(* CoDeSys 2.3.9.52 project: TrafficLights_pedeX_v1.pro *)
(* Libraries: STANDARD.LIB 16.8.17 14:08:57 *)

(* Global variable list: Global_Variables *)
VAR_GLOBAL
	I_S1		: BOOL; (*Pedestrian X button North*)
	I_S2		: BOOL; (*Pedestrian X button South*)
	O_L1_N_Red	: BOOL; (*Light red, Pedestrian North-South*)
	O_L3_N_Grn	: BOOL;	(*Light green, Pedestrian North-South*)
	O_L4_E_Red	: BOOL;	(*Light red, Cars East-West*)
	O_L5_E_Yel	: BOOL;	(*Light yellow, Cars East-West*)
	O_L6_E_Grn  	: BOOL;	(*Light green, Cars East-West*)
END_VAR

(* POU PRG_BlinkingSimple, ST *)
PROGRAM PRG_BlinkingSimple
(*Niko Siltala
Avustavia laskentaoperaatioita
- vilkutussignaalit
*)
VAR_OUTPUT
	bSign1Hz:BOOL;					(*1 Hz (60krt/min) taajudella vaihteleva signaali*)
END_VAR
VAR
	bInitDone	: BOOL	:=FALSE;	(*Ohjelman initialisointi*)
	c : INT	:=0;				(*Blink counter*)
END_VAR
(*Ohjelman initialisoinnit - Suoritetaan vain kertaalleen*)
IF NOT bInitDone THEN
	bInitDone := TRUE;
END_IF;

(*Making 1Hz blinking signal in case of simulator*)
CASE c OF
0:
	bSign1Hz:= TRUE;
1:
	bSign1Hz:= FALSE;
ELSE
	bSign1Hz:= FALSE;
END_CASE;

(*Add counter *)
c:= c + 1;
IF c > 1 THEN
	c := 0;
END_IF;
END_PROGRAM

(* POU SFC_StateModel, SFC *)
PROGRAM SFC_StateModel
VAR
	tDelay	: TIME	:= T#1s;
	tDelay_Walk : TIME := T#5s;
	srPedestrianReq	: SR;	(*Request from pedestrians has arrived*)
END_VAR
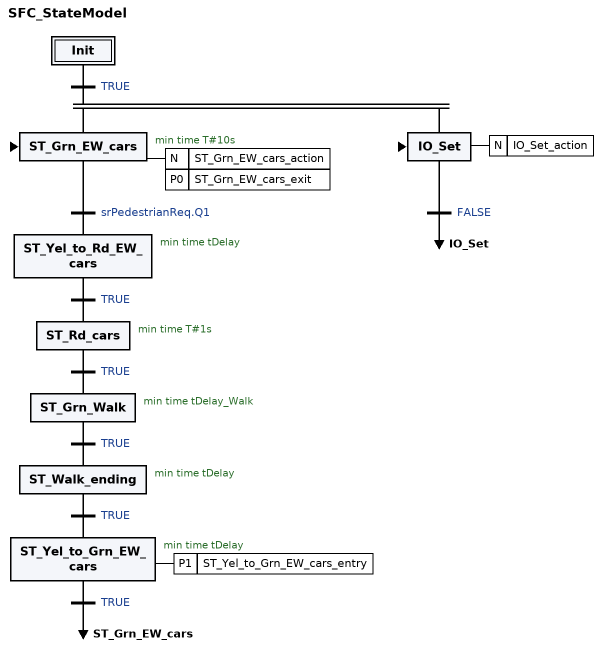
INITIAL_STEP Init:
END_STEP
TRANSITION FROM Init TO (ST_Grn_EW_cars, IO_Set) := TRUE;
END_TRANSITION
STEP ST_Grn_EW_cars: (* min time T#10s *)
	ST_Grn_EW_cars_action(N);
	ST_Grn_EW_cars_exit(P0);
END_STEP
TRANSITION FROM ST_Grn_EW_cars TO ST_Yel_to_Rd_EW_cars := srPedestrianReq.Q1;
END_TRANSITION
STEP ST_Yel_to_Rd_EW_cars: (* min time tDelay *)
END_STEP
TRANSITION FROM ST_Yel_to_Rd_EW_cars TO ST_Rd_cars := TRUE;
END_TRANSITION
STEP ST_Rd_cars: (* min time T#1s *)
END_STEP
TRANSITION FROM ST_Rd_cars TO ST_Grn_Walk := TRUE;
END_TRANSITION
STEP ST_Grn_Walk: (* min time tDelay_Walk *)
END_STEP
TRANSITION FROM ST_Grn_Walk TO ST_Walk_ending := TRUE;
END_TRANSITION
STEP ST_Walk_ending: (* min time tDelay *)
END_STEP
TRANSITION FROM ST_Walk_ending TO ST_Yel_to_Grn_EW_cars := TRUE;
END_TRANSITION
STEP ST_Yel_to_Grn_EW_cars: (* min time tDelay *)
	ST_Yel_to_Grn_EW_cars_entry(P1);
END_STEP
TRANSITION FROM ST_Yel_to_Grn_EW_cars TO ST_Grn_EW_cars := TRUE;
END_TRANSITION
STEP IO_Set:
	IO_Set_action(N);
END_STEP
TRANSITION FROM IO_Set TO IO_Set := FALSE;
END_TRANSITION

ACTION ST_Grn_EW_cars_action:
srPedestrianReq(
	SET1:= I_S1 OR I_S2,
	RESET:= FALSE,
	Q1=> );
END_ACTION

ACTION ST_Grn_EW_cars_exit:
srPedestrianReq(SET1:=FALSE , RESET:=TRUE, Q1=> );
END_ACTION

ACTION ST_Yel_to_Grn_EW_cars_entry:
srPedestrianReq(SET1:=FALSE , RESET:=TRUE, Q1=> );
END_ACTION

ACTION IO_Set_action:
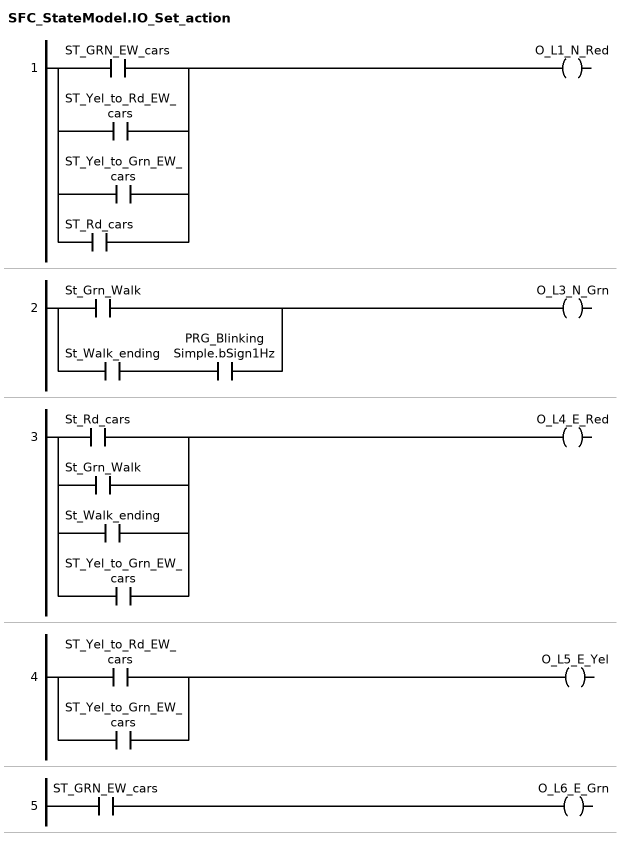
_LD_ (* Ladder Diagram *)
NETWORK 1
	{ [ST_GRN_EW_cars] | [ST_Yel_to_Rd_EW_cars] | [ST_Yel_to_Grn_EW_cars] | [ST_Rd_cars] } --- (O_L1_N_Red)
NETWORK 2
	{ [St_Grn_Walk] | [St_Walk_ending] - [PRG_BlinkingSimple.bSign1Hz] } --- (O_L3_N_Grn)
NETWORK 3
	{ [St_Rd_cars] | [St_Grn_Walk] | [St_Walk_ending] | [ST_Yel_to_Grn_EW_cars] } --- (O_L4_E_Red)
NETWORK 4
	{ [ST_Yel_to_Rd_EW_cars] | [ST_Yel_to_Grn_EW_cars] } --- (O_L5_E_Yel)
NETWORK 5
	[ST_GRN_EW_cars] --- (O_L6_E_Grn)
_END_LD_
(* the same logic as Structured Text *)
(* Network 1 *)
O_L1_N_Red := ST_GRN_EW_cars OR ST_Yel_to_Rd_EW_cars OR ST_Yel_to_Grn_EW_cars OR ST_Rd_cars;
(* Network 2 *)
O_L3_N_Grn := St_Grn_Walk OR St_Walk_ending AND PRG_BlinkingSimple.bSign1Hz;
(* Network 3 *)
O_L4_E_Red := St_Rd_cars OR St_Grn_Walk OR St_Walk_ending OR ST_Yel_to_Grn_EW_cars;
(* Network 4 *)
O_L5_E_Yel := ST_Yel_to_Rd_EW_cars OR ST_Yel_to_Grn_EW_cars;
(* Network 5 *)
O_L6_E_Grn := ST_GRN_EW_cars;
END_ACTION
END_PROGRAM

(* Visualisation VC_Main
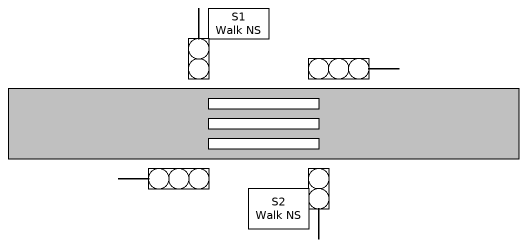
ellipse at (300,160)-(321,181): alarm colour if .O_L1_N_Red
ellipse at (300,180)-(321,201): alarm colour if .O_L3_N_Grn
rounded rectangle at (200,0)-(261,31): text "S1 / Walk NS"; alarm colour if .I_S1; taps .I_S1
rounded rectangle at (240,180)-(301,221): text "S2 / Walk NS"; alarm colour if .I_S2; taps .I_S2
ellipse at (180,160)-(201,181): alarm colour if .O_L4_E_Red
ellipse at (160,160)-(181,181): alarm colour if .O_L5_E_Yel
ellipse at (140,160)-(161,181): alarm colour if .O_L6_E_Grn
ellipse at (300,50)-(321,71): alarm colour if .O_L4_E_Red
ellipse at (320,50)-(341,71): alarm colour if .O_L5_E_Yel
ellipse at (340,50)-(361,71): alarm colour if .O_L6_E_Grn
ellipse at (180,50)-(201,71): alarm colour if .O_L1_N_Red
ellipse at (180,30)-(201,51): alarm colour if .O_L3_N_Grn
12 more shapes without text or variables
*)
